FUNCTION_BLOCK FB_Coil_Ctrl
VAR_INPUT
	i_Interlocks		:ARRAY[1..5] OF BOOL;
	i_AutoCmd			:BOOL;
	i_ManCmd			:BOOL;
	i_ServiceMode		:BOOL;
END_VAR
VAR_OUTPUT
	q_InterlocksOK		:BOOL;
	q_bCmd				:BOOL;
END_VAR
VAR
	bCmd				:BOOL;
	tofCMD				:TOF;
END_VAR

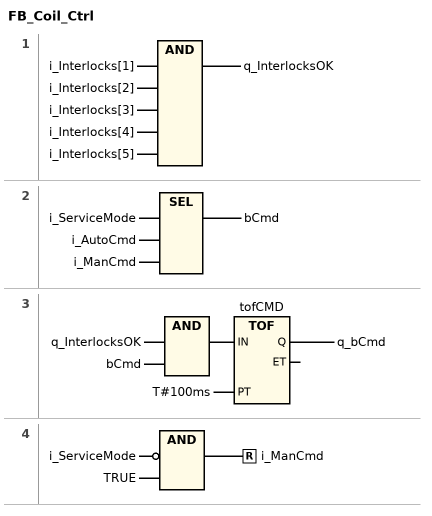
// NETWORK 1
q_InterlocksOK := i_Interlocks[1] AND i_Interlocks[2] AND i_Interlocks[3] AND i_Interlocks[4] AND i_Interlocks[5];

// NETWORK 2
bCmd := SEL(i_ServiceMode, i_AutoCmd, i_ManCmd);

// NETWORK 3
tofCMD(IN := q_InterlocksOK AND bCmd, PT := T#100ms); // TOF
q_bCmd := tofCMD.Q;

// NETWORK 4
i_ManCmd R= NOT i_ServiceMode AND TRUE;

END_FUNCTION_BLOCK

(* stored: Version 1.1.0.1, ProductVersion 3.1.4024.12
   POU FB_Coil_Ctrl: Id {8a4d27d2-3ad2-4e80-839d-2186ad87d105}, SpecialFunc None *)
